// TIA Portal V18 export
DATA_BLOCK "LowPassFilter_DB"   // DB4
// stored: InstanceOfName LowPassFilter, InstanceOfType FB
"LowPassFilter"
   // VAR_INPUT
   //    InputSignal : Real;
   //    Alpha : Real;
   // END_VAR
   // VAR_OUTPUT
   //    FilteredSignal : Real;
   // END_VAR
   // VAR
   //    LastValue : Real;
   //    AlphaInt : Real;
   // END_VAR
BEGIN
END_DATA_BLOCK
